{attribute addProperty BoxType "AT2026-0250-0020"}
{attribute addProperty Id "A_0078_AT2001_5250_0019_AT2001_5250AT2001_C5E5984862678.25"}
{attribute addProperty CRC "3620911109"}
{attribute addProperty SizeInBites "626"}
{attribute addProperty SizeInBytes "78.25"}
TYPE A_0066_AT2026_0250_0020_AT2026_0250_D7D2B805 EXTENDS AT2026_BA5A9548 :
STRUCT
	{attribute addProperty Name "A_0078_AT2001_5250_0019_AT2001_5250"}
	A_0078_AT2001_5250_0019_AT2001_5250 : AT2001_C5E59848;
END_STRUCT
END_TYPE

(* stored: Version 1.2.0.0, ProductVersion 3.1.4024.9
   DUT A_0066_AT2026_0250_0020_AT2026_0250_D7D2B805: Id {814b7344-f345-4860-80c1-61990e5fb930} *)
